(* IEC 61131-3 sources: moqui-plc/agent-skills/skills/moqui-plc-designer/references/plc-codegen-templates, 9 files *)

(* ---- DeviceFacade.template.dut ---- *)
(*
 * DeviceFacade implementation for managing devices and logical parameters.
 *
 * Naming rules:
 *   deviceName + parameterName or parameterName -> logical signal
 *   deviceName + parameterName or parameterName + Min/Max -> limits
 *
 * All digital signals (boolean) are active-high (positive logic).
 * All durations are expressed in seconds TUnit.
 *)
TYPE DeviceFacade : STRUCT
    (* ========== Analog process/environment parameters ========== *)
${ANALOG_SIGNAL_DECLARATIONS}

    (* ========== Digital process/environment parameters ========== *)
${DIGITAL_SIGNAL_DECLARATIONS}

    (* Boolean predicates - computed each scan by MainRuleEngine *)
${PREDICATE_DECLARATIONS}

    (* Operating-mode flags and process timing (mapped from recipe). *)
${PROCESS_MODE_DECLARATIONS}

    (* Main FSM state and transition request/acknowledge commands *)
    status : ${MAIN_STATUS_ENUM} := ${INITIAL_STATUS};
    lastStatus : ${MAIN_STATUS_ENUM} := ${INITIAL_STATUS};
${STATE_REQUEST_DECLARATIONS}

    (* Subsystem FSM states exposed for diagnostics and upstream publication. *)
${SUBSYSTEM_FSM_DECLARATIONS}

    (* ========== Atomic devices ========== *)
${ATOMIC_DEVICE_DECLARATIONS}

    (* Signal management - centralised fault / alarm / warning engine *)
    signalMgmt : SignalMgmt;
END_STRUCT END_TYPE

(* ---- IOFacade.template.dut ---- *)
(*
 * IOFacade implementation for managing physical devices and input/output signals/terminals.
 * Input/Output physical terminals naming rules.
 * From each value of the Parameter entity 3 signals will be generated, according to the following naming convention:
 *     deviceName + parameterName or parameterName + physicalAddress (e.g.: Channel + PhysicalAddress for Modbus)
 *     deviceName + parameterName or parameterName + Min/Max + physicalAddress (e.g.: Channel + PhysicalAddress for Modbus)
 *
 * The physicalAdddress suffix will have the following syntax:
 *    %<memory area prefix> ( <size prefix> )? <memory position>
 * where
 *    <memory area prefix> : I | Q | M
 *    <size prefix> : X | B | W | D
 *    <memory position> : <number> ( .<number> )* (* Depends on the target system *)
 *
 * An alternative is to use semantic signal naming rules.
 *)
TYPE IOFacade : STRUCT
    (* ========== Phyisical Input Terminals/Signals ========== *)
${PHYSICAL_INPUT_DECLARATIONS}

    (* ========== Phyisical Output Terminals/Signals ========== *)
${PHYSICAL_OUTPUT_DECLARATIONS}
END_STRUCT END_TYPE

(* Generation notes:
 * - This file is auto-generable from DeviceRequestItem metadata or from naming conventions.
 * - The logical-to-physical mapping remains outside this template and stays manual in V1.
 *
 * Questions for the skill/user:
 * 1. Should names come from DeviceRequestItem.requestItemName or from naming conventions?
 * 2. Which physical signals are inputs and which are outputs?
 * 3. What IEC type should be used for each signal?
 * 4. Are there address-based names, semantic names, or both?
 *)

(* ---- MainStatus.template.dut ---- *)
{attribute 'qualified_only'}
{attribute 'strict'}
TYPE MainStatus : (
${MAIN_STATUS_ITEMS}
); END_TYPE

(* Questions for the skill/user:
 * 1. Which StatusFlow is used for the main orchestration FSM?
 * 2. In which order should the states appear in the enum?
 * 3. Which state is the initial steady state?
 * 4. Which state is the fault state?
 *
 * Generation note:
 * - This enum is typically derived from StatusFlowItem entries related to the selected main StatusFlow.
 * - The generated names should match the identifiers used by Main.pou and MainRuleEngine.pou.
 *)

(* ---- SubsystemStatus.template.dut ---- *)
{attribute 'qualified_only'}
{attribute 'strict'}
TYPE ${SUBSYSTEM_STATUS_TYPE} :
(
${SUBSYSTEM_STATUS_ITEMS}
);
END_TYPE

(* ---- DeviceDiagnostics.template.pou ---- *)
{attribute 'no_assign'}
(* Device diagnostics *)
FUNCTION_BLOCK DeviceDiagnostics
VAR_EXTERNAL
    dev : DeviceFacade;
END_VAR
VAR_INPUT
    operationType : OperatingMode := OperatingMode.Run;
END_VAR
VAR_OUTPUT
    error : BOOL;
END_VAR

error := TRUE;

(* Signal management engine *)
(*
 * Prepare a fresh scan (clears the accumulated output action).
 * Then process each device signal in priority order.
 * ImmediateStop -> faultRequest := TRUE -> Main enters Fault state.
 *)
dev.signalMgmt(operationType := SignalMgmtOperatingMode.Prepare);
dev.signalMgmt.operationType := SignalMgmtOperatingMode.Process;

(* Device faults *)
${BLOCKING_DEVICE_SIGNAL_RULES}

(* Environmental / safety diagnostics *)
${SAFETY_SIGNAL_RULES}

error := FALSE;

(* Questions for the skill/user:
 * 1. Which device faults are blocking and must trigger ImmediateStop?
 * 2. For each blocking device, which signal should be monitored:
 *    fault, invalidConfig, cmdError, externalFault, etc.?
 * 3. Which environmental/safety predicates should become alarms?
 * 4. Which predicates are warnings only and should not stop the machine?
 *)

(* ---- DeviceManager.template.pou ---- *)
{attribute 'no_assign'}
(* Hardware Abstraction Layer (HAL) orchestrator.
 *
 * Drives all physical device FBs once per scan.
 * Main component sets the enable/disable request flags; DeviceManager wires them
 * to the individual Actuator / ProcessPid FBs.
 *
 * Call order within the PLC task:
 *   InputSignalUpdate (updates feedback signals from field)
 *   Main (FSM + DeviceRuleEngine -> sets request flags)
 *   DeviceManager (this block - drives device FBs)
 *   OutputSignalUpdate (maps device outputs to physical terminals)
 *
 * Handshake note (Actuator FBs):
 *   enableRequest / disableRequest are VAR_IN_OUT.  The Actuator FB clears
 *   the flag as its acknowledgment.  Main.pou re-asserts the flag each scan
 *   from dev.xxxEnableRequest, so the handshake is level-triggered.
 *
 * ProcessPid note (ahuFan):
 *   ProcessPid uses a plain BOOL 'enable' input - no VAR_IN_OUT handshake.
 *   Setting enable := FALSE ramps the output to 0 and disables the controller.
 *)
FUNCTION_BLOCK DeviceManager
VAR_EXTERNAL
    clks : Clocks;
    dev : DeviceFacade;
END_VAR
VAR_INPUT
    operationType : OperatingMode := OperatingMode.Run;
END_VAR

(* Atomic device orchestration *)
${DEVICE_MANAGER_CALLS}

(* Questions for the skill/user:
 * 1. Which atomic devices must be called every scan?
 * 2. For each Actuator, which enableRequest/disableRequest flags drive it?
 * 3. For each ProcessPid, which enable/setpoint/feedback signals drive it?
 * 4. For each Axis or AxisGroup, which command/enable structures are used?
 *)

(* ---- Main.template.pou ---- *)
{attribute 'no_assign'}
(*
 * NOTE: In general, the Main component implements the control logic of automated industrial systems (Finite State Machine - FSM)
 * using hierarchical control architectures. It separates control policies from implementation mechanisms,
 * and diagnostic mechanisms from failure/error reaction and system reset policies.
 *
 * MainRuleEngine generates transition requests; Main consumes them.
 * DeviceManager orchestrates the individual device FBs.
 *
 * Call order in the PLC task:
 *   InputSignalUpdate -> Main -> DeviceManager -> OutputSignalUpdate
 *)
FUNCTION_BLOCK Main
VAR_EXTERNAL
    dev : DeviceFacade;
    workEffort : WorkEffort;
END_VAR
VAR_INPUT
    operationType : OperatingMode;
    enable : BOOL;
END_VAR
VAR_OUTPUT
    done : BOOL;
    error : BOOL;
END_VAR
VAR CONSTANT
    componentName : STRING := '${COMPONENT_NAME}';
END_VAR
VAR
    (* Logger facade *)
    logger : LoggerFacade;
    (* FSM transition logic *)
    ruleEngine : MainRuleEngine;
    (* Optional: define one or more FSMs for managing subsystems, if needed *)
    (* HAL manager *)
    deviceManager : DeviceManager;
END_VAR

(* Logger facade init *)
logger.enable := TRUE; logger.loggerName := componentName;

IF NOT enable THEN RETURN; END_IF

(* Init: device setup and configuration *)
IF (operationType = OperatingMode.Init) THEN
    logger(message := 'Setup and configuration of all devices.', level := LogLevel.DEBUG);
    (* The static device configuration parameters are mapped directly by the device config manager (recipe manager),
     * while only the dynamic parameters are mapped below in the standby status.
     *)
    (* Reset signal manager *)
    dev.signalMgmt(operationType := SignalMgmtOperatingMode.Reset, loggerName := componentName);
    dev.status := ${INITIAL_STATUS};
    dev.lastStatus := ${INITIAL_STATUS};
    done := FALSE;
${INIT_ASSIGNMENTS}
ELSE
    (* FSM transition-condition rule engine *)
    logger(message := 'Run FSM transition-condition logic.', level := LogLevel.DEBUG);
    ruleEngine(operationType := operationType);
END_IF;

dev.lastStatus := dev.status;

(* Fault overrides any other state *)
IF dev.faultRequest THEN dev.status := ${FAULT_STATUS}; END_IF;

(* Main FSM - Output function + State-update function *)
logger(message := 'Run Main FSM.', level := LogLevel.DEBUG);
CASE dev.status OF
${MAIN_FSM_CASE_BLOCKS}
END_CASE;

done := dev.isCompleted;

(* Device orchestration (HAL) *)
logger(message := 'Update devices.', level := LogLevel.DEBUG);
deviceManager(operationType := operationType);

(* Questions for the skill/user:
 * 1. Which StatusFlow drives this Main FSM?
 * 2. What is the initial state and what is the fault state?
 * 3. For each state, which output requests must be asserted or cleared?
 * 4. For each state, which next-state requests may be consumed here?
 *)

(* ---- MainRuleEngine.template.pou ---- *)
{attribute 'no_assign'}
(*
 * MainRuleEngine - transition-condition logic for the supervisor FSM.
 *
 * Responsibilities:
 *   1. Reset transition requests to safe defaults.
 *   2. Run the signal management engine (fault / alarm / warning detection).
 *   3. Compute boolean predicates from sensor feedback and recipe setpoints.
 *   4. Implement the per-state transition-condition rules.
 *
 * Default / persistence convention
 * At the top of every scan standbyRequest is set TRUE (safe default).
 * Each ACTIVE-state CASE block MUST:
 *   - Set standbyRequest := FALSE (keep current state) in the ELSE branch.
 *   - Set standbyRequest := TRUE (or leave as-is) when an EXIT condition is met.
 *   - Set standbyRequest := FALSE and another*Request := TRUE to switch phase.
 *
 * Without the ELSE branch the system would exit any active state to Standby
 * on the very first scan - a single-scan flash rather than a persistent phase.
 *)
FUNCTION_BLOCK MainRuleEngine
VAR_EXTERNAL
    clks : Clocks;
    dev : DeviceFacade;
    workEffort : WorkEffort;
END_VAR
VAR_INPUT
    operationType : OperatingMode := OperatingMode.Run;
END_VAR
VAR_OUTPUT
    error : BOOL;
END_VAR
VAR
    (* Device diagnostics *)
    deviceDiags : DeviceDiagnostics;
END_VAR

(* Reset transition requests to safe defaults.
 *
 * standbyRequest = TRUE  -> return to / stay in Standby (safe default).
 * Active-state CASE blocks override to FALSE to keep the current phase alive,
 * or set another *Request to switch phases.
 *)
${REQUEST_RESET_BLOCK}

deviceDiags(operationType := operationType, error => error);

(* Compute sensor predicates *)
${SENSOR_PREDICATES}

(* Process timing - generic run / break cycle *)
IF clks.clock1s THEN
    dev.processActualDuration := dev.processActualDuration + 1;

    IF dev.timeBreakEnabled AND dev.status = ${BREAK_STATUS} THEN
        dev.actualBreakDuration := dev.actualBreakDuration + 1;
        IF dev.estimatedBreakDuration > 0 THEN
            IF (dev.actualBreakDuration >= dev.estimatedBreakDuration)
                    AND (dev.actualBreakDuration >= dev.minBreakDuration) THEN
                dev.timeBreakEnabled := FALSE;
                dev.actualRuntime := 0;
                dev.actualBreakDuration := 0;
            END_IF;
        END_IF;
    ELSE
        dev.actualRuntime := dev.actualRuntime + 1;
        IF dev.estimatedRuntime > 0 THEN
            dev.processRemainingDuration := dev.processEstimatedDuration - dev.processActualDuration;
            IF NOT dev.timeBreakEnabled
                    AND (dev.actualRuntime >= dev.estimatedRuntime)
                    AND (dev.actualRuntime >= dev.minRuntime) THEN
                dev.timeBreakEnabled := TRUE;
                dev.actualBreakDuration := 0;
            END_IF;
        END_IF;
    END_IF;

    IF dev.processEstimatedDuration > 0 THEN
        dev.isCompleted :=
            (dev.processActualDuration >= dev.processEstimatedDuration)
            AND (dev.processActualDuration >= dev.processMinDuration);
    END_IF;
END_IF;

(* Fault gate *)
IF error OR ((dev.signalMgmt.cumulativeOutputAction AND SignalOutputAction.ImmediateStop) <> 0) THEN
    dev.faultRequest := TRUE;
    RETURN;
END_IF;

(* Transition-condition rule engine
 *
 * Persistence rule: every active-state CASE MUST end with
 *   ELSE dev.standbyRequest := FALSE; (* keep current state alive *)
 * to prevent the scan-level default (standbyRequest=TRUE) from immediately
 * bouncing the FSM back to Standby before the exit condition is reached.
 *)
CASE dev.status OF
${STATE_TRANSITION_CASES}
END_CASE;

(* Questions for the skill/user:
 * 1. Which predicates must be computed from analog/digital signals?
 * 2. Which predicates are process predicates and which are safety predicates?
 * 3. Which predicates can be inferred from existing parameter names, thresholds, hysteresis values, or seed-data rows?
 * 4. For each StatusFlowTransition, what is the boolean condition from current state to next state?
 * 5. Which transition has precedence if multiple conditions are true?
 * 6. Is the generic run/break timing block valid as-is, or does it require extension?
 *)

(* ---- SubsystemController.template.pou ---- *)
{attribute 'no_assign'}
(* Subsystem controller generated from reviewed FSM survey data. *)
FUNCTION_BLOCK ${SUBSYSTEM_CONTROLLER_TYPE}
VAR_EXTERNAL
    dev : DeviceFacade;
END_VAR
VAR_INPUT
    operationType : OperatingMode := OperatingMode.Init;
    enable : BOOL := TRUE;
END_VAR
VAR CONSTANT
    componentName : STRING := '${SUBSYSTEM_COMPONENT_NAME}';
END_VAR
VAR
    logger : LoggerFacade;
END_VAR

logger.enable := TRUE; logger.loggerName := componentName;

IF operationType = OperatingMode.Init THEN
    dev.${SUBSYSTEM_STATUS_FIELD} := ${SUBSYSTEM_STATUS_TYPE}.${SUBSYSTEM_INITIAL_STATUS};
    dev.${SUBSYSTEM_LAST_STATUS_FIELD} := ${SUBSYSTEM_STATUS_TYPE}.${SUBSYSTEM_INITIAL_STATUS};
    RETURN;
END_IF;

IF NOT enable THEN RETURN; END_IF;

dev.${SUBSYSTEM_LAST_STATUS_FIELD} := dev.${SUBSYSTEM_STATUS_FIELD};
${SUBSYSTEM_PREDICATE_ASSIGNMENTS}
CASE dev.${SUBSYSTEM_STATUS_FIELD} OF
${SUBSYSTEM_CASE_BLOCKS}
END_CASE;
END_FUNCTION_BLOCK
